// TIA Portal V17 export
// export: Created 2024-09-02T12:50:25.6748538Z, ExportSetting WithDefaults, DisplayName Totally Integrated Automation Portal, DisplayVersion V17, DisplayName TIA Portal Openness, DisplayVersion V17, DisplayName TIA Portal Version Control Interface, DisplayVersion V17, DisplayName STEP 7 Professional, DisplayVersion V17, DisplayName STEP 7 Safety, DisplayVersion V17, DisplayName WinCC Professional, DisplayVersion V17
VAR_GLOBAL   // PLC tag table "OP70_1"
   IW_RFID_SLG1_OP70_1 AT %IW2002 : Word;   // Balluff BIS V Reader 1 (+M01-BX600)
   I_MM140_Y_Axis_Gripper_Front_OP70_2 AT %I53.6 : Bool;
   I_MM110_Sliding_Damper_Cap_Back_OP70_1 AT %I52.4 : Bool;
   I_MM110_Sliding_Damper_Cap_Front_OP70_1 AT %I52.5 : Bool;
   I_MM110_Damper_Cap_Present_OP70_1 AT %I52.6 : Bool;
   I_MM120_Sliding_Ball_Back_OP70_1 AT %I53.0 : Bool;
   I_MM120_Sliding_Ball_Front_OP70_1 AT %I53.1 : Bool;
   I_MM120_Ball_Present_OP70_1 AT %I53.2 : Bool;
   I_MM130_Press_Damper_UP_OP70_1 AT %I53.3 : Bool;
   "I_MM30/31_index_down_OP70_1" AT %I51.0 : Bool;
   I_Air_pressure_OK_OP70 AT %I50.7 : Bool;   // Pneumatikdruck IO (+M01-BP50.7)
   "I_MM30/31_index_up_OP70_1" AT %I51.1 : Bool;
   I_MM10_prestopper_Close_OP70_1 AT %I50.0 : Bool;   // MB10 Vorstopper geschlossen (+M01-BG50.0)
   I_MM20_stopper_close_OP70_1 AT %I50.1 : Bool;   // MB20 Stopper 1 geschlossen (+M01-BG51.0)
   I_MM10_pallet_at_prestopper_OP70_1 AT %I50.2 : Bool;   // MB10 WT am Vorstopper (+M01-BG50.1)
   I_MM20_pallet_at_stopper_OP70_1 AT %I50.3 : Bool;   // MB20 WT am Stopper 1 (+M01-BG51.1)
   Q_MM10_prestopper_open_OP70_1 AT %Q80.0 : Bool;
   Q_MM20_Stopper_open_OP70_1 AT %Q80.2 : Bool;
   "Q_MM30/31_index_Upward_OP70_1" AT %Q81.0 : Bool;
   "Q_MM30/31_index_Downward_OP70_1" AT %Q81.1 : Bool;
   Q_MM110_Sliding_Damper_Cap_Forward_OP70_1 AT %Q86.0 : Bool;
   Q_MM110_Sliding_Damper_Cap_Backward_OP70_1 AT %Q86.1 : Bool;
   Q_MM120_Sliding_Ball_Forward_OP70_1 AT %Q86.2 : Bool;
   Q_MM120_Sliding_Ball_Backward_OP70_1 AT %Q86.3 : Bool;
   Q_MM130_Press_Damper_Downward_OP70_1 AT %Q87.0 : Bool;
   Q_MM130_Press_Damper_Upward_OP70_1 AT %Q87.1 : Bool;
   QW_RFID_SLG1_OP70_1 AT %QW2002 : Word;   // Balluff BIS V Reader 1 (+M01-BX600)
END_VAR
